// TwinCAT 3 PLC project AICodesAndValidation
// Title: AI Codes And Validation
// Company: Marden Edwards
// Author: Wiktor Pytka
// ProjectVersion: 1.0.0.0
// ProgramVersion: 3.1.4026.19
// libraries:
//   Tc2_Standard, * (Beckhoff Automation GmbH)
//   Tc2_System, * (Beckhoff Automation GmbH)
// project tree:
//   DUTs/AI Codes And Validation/ E_CodeAI.TcDUT (not stored), E_CodeType.TcDUT (not stored), ST_CodeInfo.TcDUT, ST_CodeValidation.TcDUT (not stored)
//   POUs/AI Codes And Validation FBs/ FB_ClearCodeInfo.TcPOU (not stored), FB_ValidateExplicitCode.TcPOU (not stored), F_AssignValToStringWithPrefix.TcPOU (not stored), F_GetItemAI.TcPOU (not stored)
//   POUs/Utilities/ F_StringAddPrefix.TcPOU
//   Version/ Global_Version.TcGVL

// ---- DUTs/AI Codes And Validation/ST_CodeInfo.TcDUT
TYPE ST_CodeInfo :
STRUCT
	eCodeType					:	E_CodeType;

	nMinLength					: 	INT;
	nEntireLength				:	INT;
	bValidateEntireLength		: 	BOOL;
	nNumberOfAIs				:	INT;

	stGTIN 						:	ST_CodeValidation	:=		(sFieldName :='GTIN',					bNameEditable := FALSE, 		nGS1_AI := 1);
	stBatchID 					:	ST_CodeValidation	:=		(sFieldName :='BatchID', 				bNameEditable := FALSE, 		nGS1_AI := 10);
	stSerialCode 				:	ST_CodeValidation	:=		(sFieldName :='SerialCode', 			bNameEditable := FALSE, 		nGS1_AI := 21);
	stProductionOrder 			:	ST_CodeValidation	:=		(sFieldName :='ProductionOrder', 		bNameEditable := FALSE, 		nGS1_AI := 91);
	stCryptoCode				:	ST_CodeValidation	:=		(sFieldName :='CryptoCode', 			bNameEditable := FALSE, 		nGS1_AI := 93);
	stRSKU						:	ST_CodeValidation	:=		(sFieldName :='RSKU', 					bNameEditable := FALSE, 		nGS1_AI := 240);
	stMRP		 				:	ST_CodeValidation	:=		(sFieldName :='MRP', 					bNameEditable := FALSE, 		nGS1_AI := 8005);
	stBrandSpecification		:	ST_CodeValidation	:=		(sFieldName :='BrandSpec',				bNameEditable := FALSE, 		nGS1_AI := 92);
	stProduceDate				:	ST_CodeValidation	:=		(sFieldName :='ProduceDate',			bNameEditable := TRUE, 			nGS1_AI := 94);
	stUserField3				:	ST_CodeValidation	:=		(sFieldName :='',						bNameEditable := TRUE, 			nGS1_AI := 95);

END_STRUCT
END_TYPE

// ---- Version/Global_Version.TcGVL
{attribute 'TcGenerated'}
{attribute 'no-analysis'}
{attribute 'linkalways'}
// This function has been automatically generated from the project information.
VAR_GLOBAL CONSTANT
	{attribute 'const_non_replaced'}
	stLibVersion_AI_Codes_And_Validation : ST_LibVersion := (iMajor := 1, iMinor := 0, iBuild := 0, iRevision := 0, sVersion := '1.0.0.0');
END_VAR

// ---- POUs/Utilities/F_StringAddPrefix.TcPOU
(* add specified char(s) in front of a string to make up to specified length *)
FUNCTION F_StringAddPrefix : T_MaxString
VAR_INPUT
	sString		: T_MaxString;	(* initial string *)
	nTargetLen 		: UINT;			(* string length required *)
	sChar			: STRING(1);	(* char to be appended to string *)
END_VAR
VAR
	nStringLen		: UINT;
	nCharsReq		: uINT;
END_VAR
(*
-------------------------------------------------------------------------------------------------
Date		Version	Author	Comments
-------------------------------------------------------------------------------------------------
30/01/2015	3.00.00	PB		Initial release

-------------------------------------------------------------------------------------------------
*)

(* length of input string *)
nStringLen := TO_UINT(LEN(sString));

(* Chekck target string is longer than processing string *)
IF nTargetLen >= nStringLen THEN
	
	(* total prefix chars required *)
	nCharsReq := MIN(nTargetLen, SIZEOF(F_StringAddPrefix) - 1) - nStringLen;

	(* string needs additional chars *)
	IF nCharsReq > 0 THEN
	
		(* set prefix chars to specified character *)
		MEMSET(ADR(F_StringAddPrefix), F_ToASC(sChar), nCharsReq);
	
		(* append strString to output string *)
		MEMMOVE(ADR(F_StringAddPrefix) + nCharsReq, ADR(sString), nStringLen);
	
		(* reset last char to 16#00 to terminate the string *)
		MEMSET(ADR(F_StringAddPrefix) + nCharsReq + nStringLen, 16#00, 1);
	
	(* no additional chars required *)
	ELSE
	
		(* copy strString to output *)
		F_StringAddPrefix := sString;
	END_IF
ELSE
	(* copy shrinced strString to output *)
	F_StringAddPrefix := LEFT(sString, TO_INT(nTargetLen));
END_IF

END_FUNCTION
